{attribute 'qualified_only'}
{attribute 'strict'}
TYPE eEarthingSystems :
(
	None 		:= 0,	
	TN			:= 1,
	TN_ext		:= 2,
	IT			:= 3		
);
END_TYPE

(* stored: Version 1.1.0.1, ProductVersion 3.1.4026.18
   DUT eEarthingSystems: Id {1e3c194c-327c-4225-b0ec-04d0c1a04abb} *)
